Staubli VAL3: onF4Event.pgx

program onF4Event(bool& x_bSave[] (dimensions=1))
  local string l_sMessage
  local num l_nActual
  local num l_nOldValue
  local num l_nX
  local num l_nY
begin
  // look if the bButton is enable
  if bButton[3]
    //
    //
    //
  endIf
end
